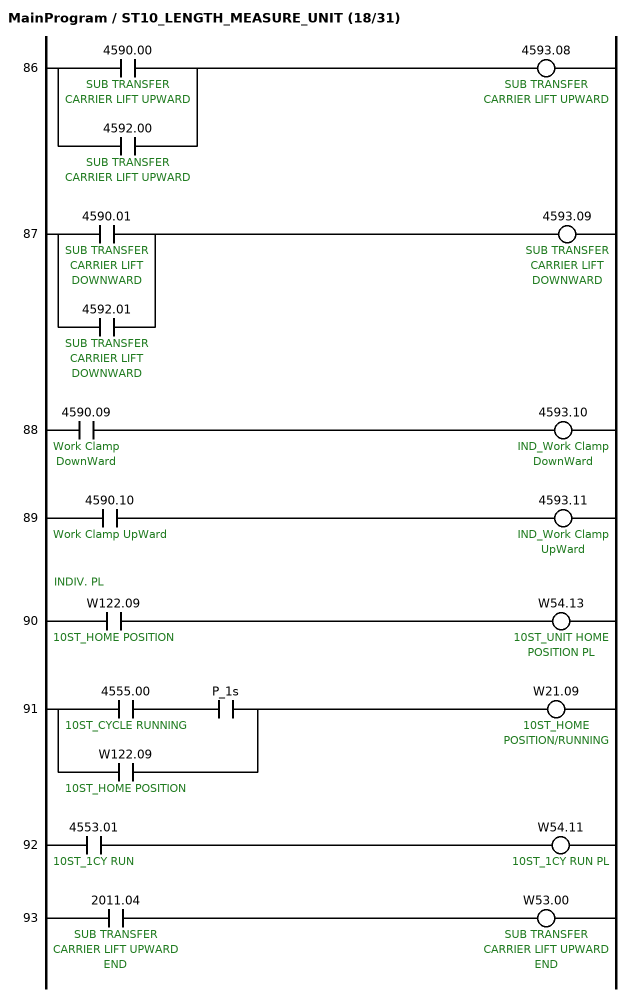
; [picture p504: MainProgram / ST10_LENGTH_MEASURE_UNIT, rungs 86-93]
; rung 86
LD 4590.00  ; SUB TRANSFER CARRIER LIFT UPWARD
OR 4592.00  ; SUB TRANSFER CARRIER LIFT UPWARD
OUT 4593.08  ; SUB TRANSFER CARRIER LIFT UPWARD
; rung 87
LD 4590.01  ; SUB TRANSFER CARRIER LIFT DOWNWARD
OR 4592.01  ; SUB TRANSFER CARRIER LIFT DOWNWARD
OUT 4593.09  ; SUB TRANSFER CARRIER LIFT DOWNWARD
; rung 88
LD 4590.09  ; Work Clamp DownWard
OUT 4593.10  ; IND_Work Clamp DownWard
; rung 89
LD 4590.10  ; Work Clamp UpWard
OUT 4593.11  ; IND_Work Clamp UpWard
; rung 90: INDIV. PL
LD W122.09  ; 10ST_HOME POSITION
OUT W54.13  ; 10ST_UNIT HOME POSITION PL
; rung 91
LD 4555.00  ; 10ST_CYCLE RUNNING
AND P_1s
OR W122.09  ; 10ST_HOME POSITION
OUT W21.09  ; 10ST_HOME POSITION/RUNNING
; rung 92
LD 4553.01  ; 10ST_1CY RUN
OUT W54.11  ; 10ST_1CY RUN PL
; rung 93
LD 2011.04  ; SUB TRANSFER CARRIER LIFT UPWARD END
OUT W53.00  ; SUB TRANSFER CARRIER LIFT UPWARD END

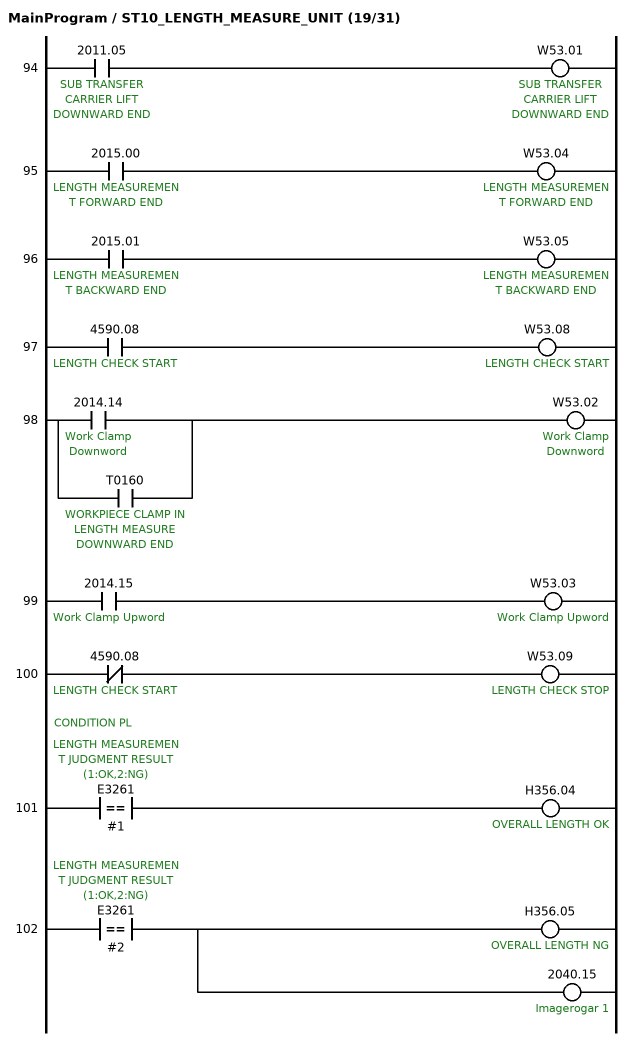
; rung 94
LD 2011.05  ; SUB TRANSFER CARRIER LIFT DOWNWARD END
OUT W53.01  ; SUB TRANSFER CARRIER LIFT DOWNWARD END
; rung 95
LD 2015.00  ; LENGTH MEASUREMENT FORWARD END
OUT W53.04  ; LENGTH MEASUREMENT FORWARD END
; rung 96
LD 2015.01  ; LENGTH MEASUREMENT BACKWARD END
OUT W53.05  ; LENGTH MEASUREMENT BACKWARD END
; rung 97
LD 4590.08  ; LENGTH CHECK START
OUT W53.08  ; LENGTH CHECK START
; rung 98
LD 2014.14  ; Work Clamp Downword
OR T0160  ; WORKPIECE CLAMP IN LENGTH MEASURE DOWNWARD END
OUT W53.02  ; Work Clamp Downword
; rung 99
LD 2014.15  ; Work Clamp Upword
OUT W53.03  ; Work Clamp Upword
; rung 100
LDNOT 4590.08  ; LENGTH CHECK START
OUT W53.09  ; LENGTH CHECK STOP
; rung 101: CONDITION PL
LD=(300) E3261 #1  ; LENGTH MEASUREMENT JUDGMENT RESULT (1:OK,2:NG)
OUT H356.04  ; OVERALL LENGTH OK
; rung 102
LD=(300) E3261 #2  ; LENGTH MEASUREMENT JUDGMENT RESULT (1:OK,2:NG)
OUT H356.05  ; OVERALL LENGTH NG
OUT 2040.15  ; Imagerogar 1

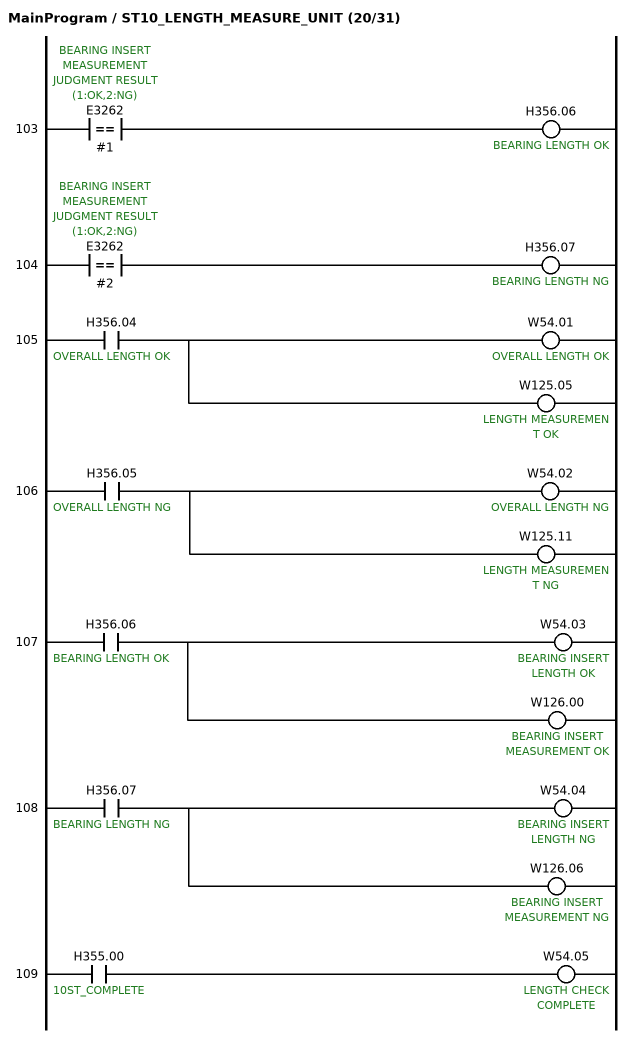
; rung 103
LD=(300) E3262 #1  ; BEARING INSERT MEASUREMENT  JUDGMENT RESULT (1:OK,2:NG)
OUT H356.06  ; BEARING LENGTH OK
; rung 104
LD=(300) E3262 #2  ; BEARING INSERT MEASUREMENT  JUDGMENT RESULT (1:OK,2:NG)
OUT H356.07  ; BEARING LENGTH NG
; rung 105
LD H356.04  ; OVERALL LENGTH OK
OUT W54.01  ; OVERALL LENGTH OK
OUT W125.05  ; LENGTH MEASUREMENT OK
; rung 106
LD H356.05  ; OVERALL LENGTH NG
OUT W54.02  ; OVERALL LENGTH NG
OUT W125.11  ; LENGTH MEASUREMENT NG
; rung 107
LD H356.06  ; BEARING LENGTH OK
OUT W54.03  ; BEARING INSERT LENGTH OK
OUT W126.00  ; BEARING INSERT MEASUREMENT OK
; rung 108
LD H356.07  ; BEARING LENGTH NG
OUT W54.04  ; BEARING INSERT LENGTH NG
OUT W126.06  ; BEARING INSERT MEASUREMENT NG
; rung 109
LD H355.00  ; 10ST_COMPLETE
OUT W54.05  ; LENGTH CHECK COMPLETE

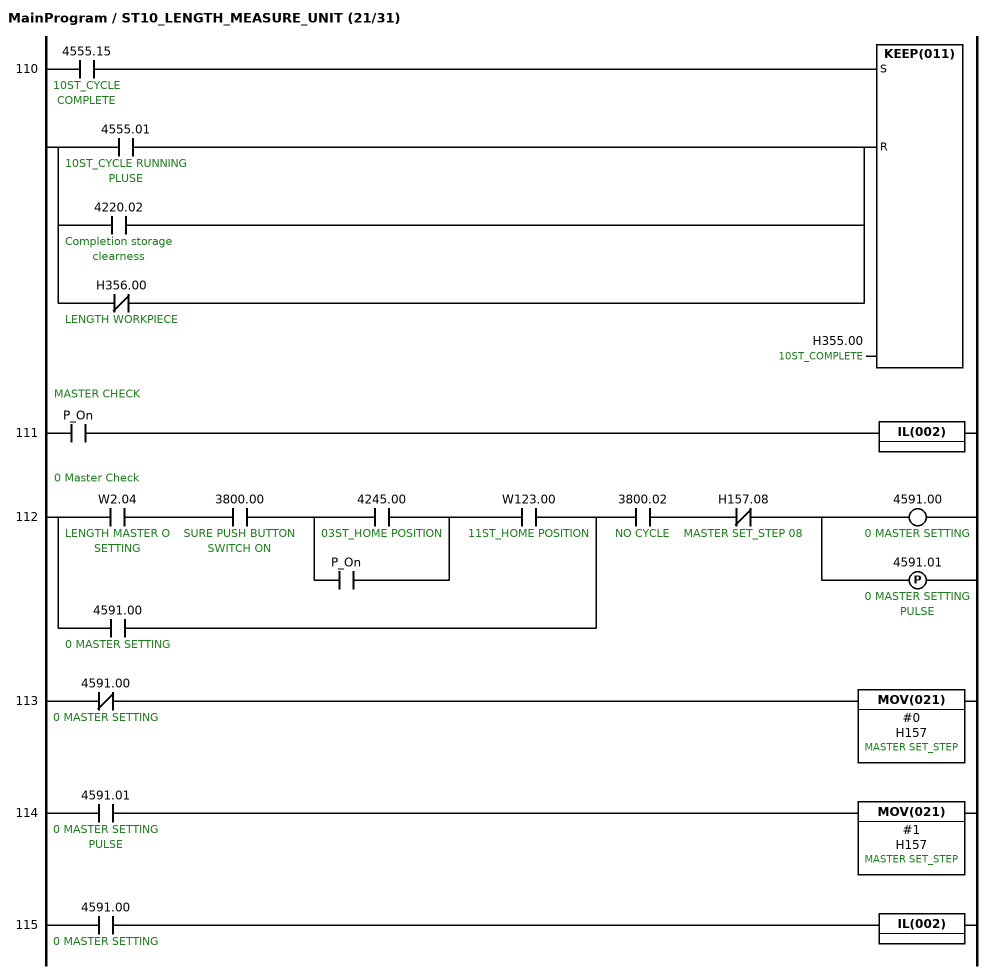
; rung 110
LD 4555.15  ; 10ST_CYCLE COMPLETE
LD 4555.01  ; 10ST_CYCLE RUNNING PLUSE
OR 4220.02  ; Completion storage clearness
ORNOT H356.00  ; LENGTH WORKPIECE
KEEP(011) H355.00  ; 10ST_COMPLETE
; rung 111: MASTER CHECK
LD P_On
IL(002)
; rung 112: 0 Master Check
LD W2.04  ; LENGTH MASTER O SETTING
AND 3800.00  ; SURE PUSH BUTTON SWITCH ON
LD 4245.00  ; 03ST_HOME POSITION
OR P_On
ANDLD
AND W123.00  ; 11ST_HOME POSITION
OR 4591.00  ; 0 MASTER SETTING
AND 3800.02  ; NO CYCLE
ANDNOT H157.08  ; MASTER SET_STEP 08
OUT 4591.00  ; 0 MASTER SETTING
DIFU(013) 4591.01  ; 0 MASTER SETTING PULSE
; rung 113
LDNOT 4591.00  ; 0 MASTER SETTING
MOV(021) #0 H157  ; MASTER SET_STEP
; rung 114
LD 4591.01  ; 0 MASTER SETTING PULSE
MOV(021) #1 H157  ; MASTER SET_STEP
; rung 115
LD 4591.00  ; 0 MASTER SETTING
IL(002)

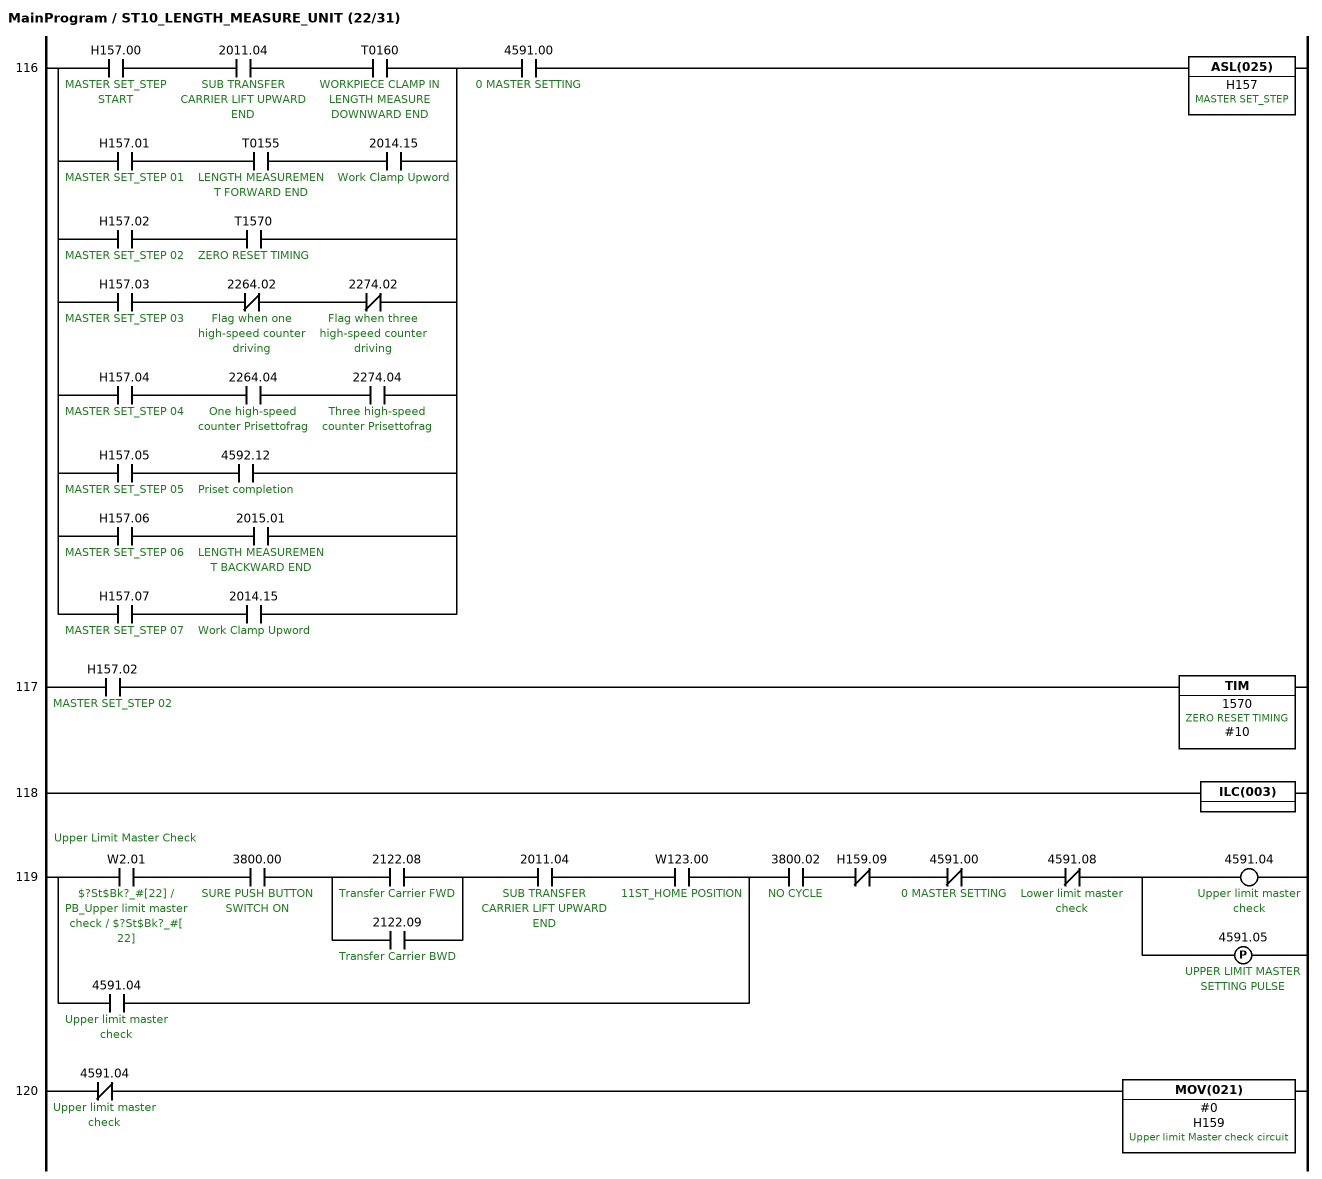
; rung 116
LD H157.00  ; MASTER SET_STEP START
AND 2011.04  ; SUB TRANSFER CARRIER LIFT UPWARD END
AND T0160  ; WORKPIECE CLAMP IN LENGTH MEASURE DOWNWARD END
LD H157.01  ; MASTER SET_STEP 01
AND T0155  ; LENGTH MEASUREMENT FORWARD END
AND 2014.15  ; Work Clamp Upword
ORLD
LD H157.02  ; MASTER SET_STEP 02
AND T1570  ; ZERO RESET TIMING
ORLD
LD H157.03  ; MASTER SET_STEP 03
ANDNOT 2264.02  ; Flag when one high-speed counter driving
ANDNOT 2274.02  ; Flag when three high-speed counter driving
ORLD
LD H157.04  ; MASTER SET_STEP 04
AND 2264.04  ; One high-speed counter Prisettofrag
AND 2274.04  ; Three high-speed counter Prisettofrag
ORLD
LD H157.05  ; MASTER SET_STEP 05
AND 4592.12  ; Priset completion
ORLD
LD H157.06  ; MASTER SET_STEP 06
AND 2015.01  ; LENGTH MEASUREMENT BACKWARD END
ORLD
LD H157.07  ; MASTER SET_STEP 07
AND 2014.15  ; Work Clamp Upword
ORLD
AND 4591.00  ; 0 MASTER SETTING
ASL(025) H157  ; MASTER SET_STEP
; rung 117
LD H157.02  ; MASTER SET_STEP 02
TIM 1570 #10  ; ZERO RESET TIMING
; rung 118
ILC(003)
; rung 119: Upper Limit Master Check
LD W2.01  ; $?St$Bk?_#[22] / PB_Upper limit master check / $?St$Bk?_#[22]
AND 3800.00  ; SURE PUSH BUTTON SWITCH ON
LD 2122.08  ; Transfer Carrier FWD
OR 2122.09  ; Transfer Carrier BWD
ANDLD
AND 2011.04  ; SUB TRANSFER CARRIER LIFT UPWARD END
AND W123.00  ; 11ST_HOME POSITION
OR 4591.04  ; Upper limit master check
AND 3800.02  ; NO CYCLE
ANDNOT H159.09
ANDNOT 4591.00  ; 0 MASTER SETTING
ANDNOT 4591.08  ; Lower limit master check
OUT 4591.04  ; Upper limit master check
DIFU(013) 4591.05  ; UPPER LIMIT MASTER SETTING PULSE
; rung 120
LDNOT 4591.04  ; Upper limit master check
MOV(021) #0 H159  ; Upper limit Master check circuit

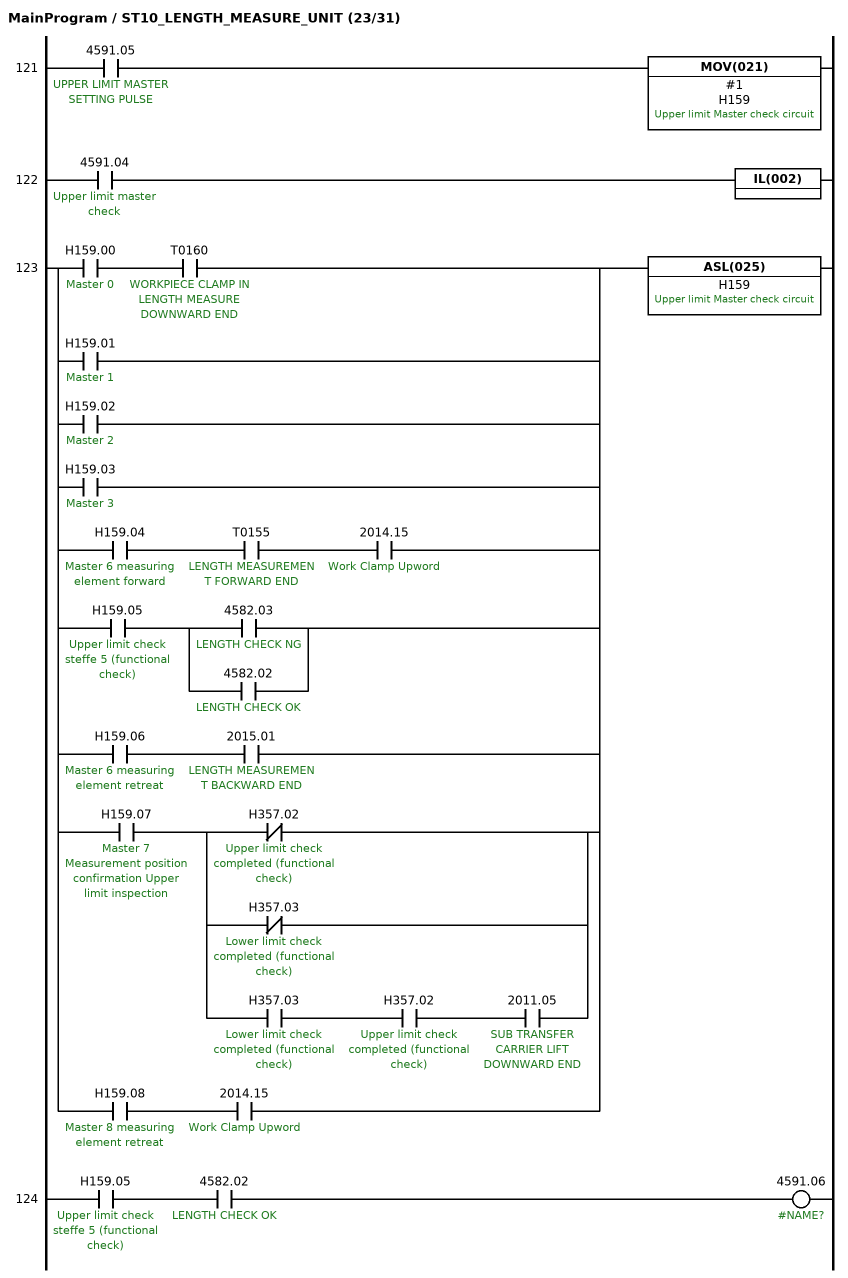
; rung 121
LD 4591.05  ; UPPER LIMIT MASTER SETTING PULSE
MOV(021) #1 H159  ; Upper limit Master check circuit
; rung 122
LD 4591.04  ; Upper limit master check
IL(002)
; rung 123
LD H159.00  ; Master 0
AND T0160  ; WORKPIECE CLAMP IN LENGTH MEASURE DOWNWARD END
OR H159.01  ; Master 1
OR H159.02  ; Master 2
OR H159.03  ; Master 3
LD H159.04  ; Master 6 measuring element forward
AND T0155  ; LENGTH MEASUREMENT FORWARD END
AND 2014.15  ; Work Clamp Upword
ORLD
LD H159.05  ; Upper limit check steffe 5 (functional check)
LD 4582.03  ; LENGTH CHECK NG
OR 4582.02  ; LENGTH CHECK OK
ANDLD
ORLD
LD H159.06  ; Master 6 measuring element retreat
AND 2015.01  ; LENGTH MEASUREMENT BACKWARD END
ORLD
LD H159.07  ; Master 7 Measurement position confirmation Upper limit inspection
LDNOT H357.02  ; Upper limit check completed (functional check)
ORNOT H357.03  ; Lower limit check completed (functional check)
LD H357.03  ; Lower limit check completed (functional check)
AND H357.02  ; Upper limit check completed (functional check)
AND 2011.05  ; SUB TRANSFER CARRIER LIFT DOWNWARD END
ORLD
ANDLD
ORLD
LD H159.08  ; Master 8 measuring element retreat
AND 2014.15  ; Work Clamp Upword
ORLD
ASL(025) H159  ; Upper limit Master check circuit
; rung 124
LD H159.05  ; Upper limit check steffe 5 (functional check)
AND 4582.02  ; LENGTH CHECK OK
OUT 4591.06  ; #NAME?

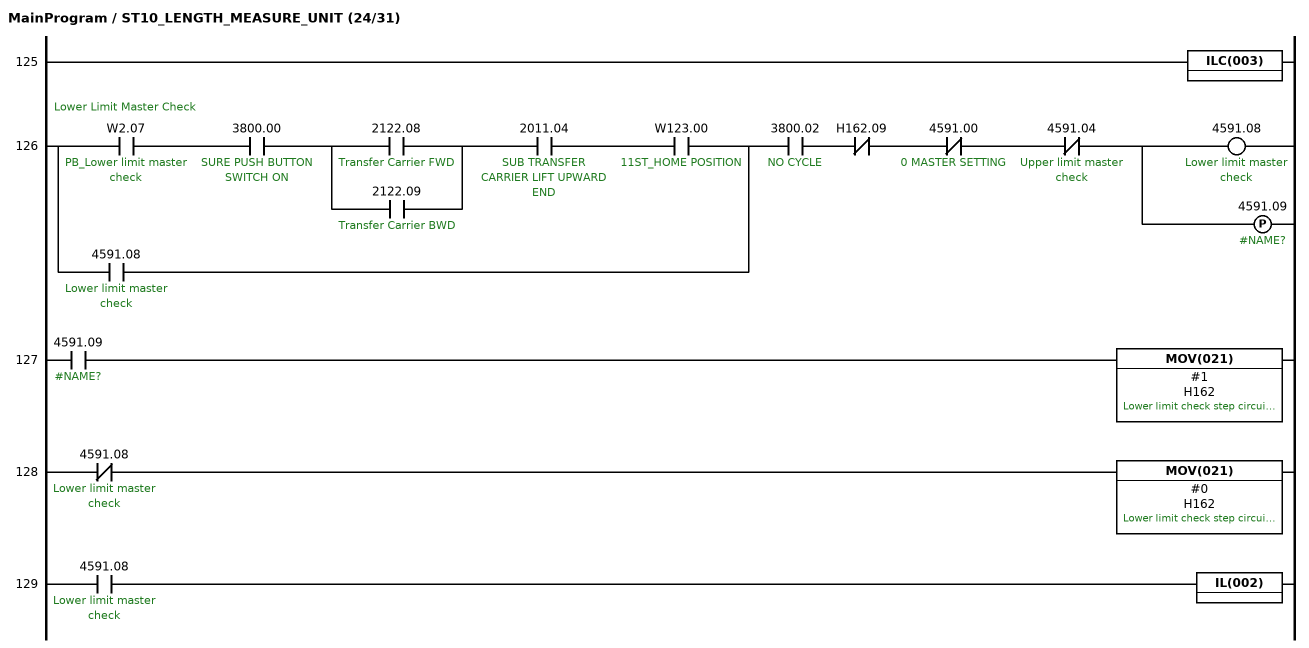
; rung 125
ILC(003)
; rung 126: Lower Limit Master Check
LD W2.07  ; PB_Lower limit master check
AND 3800.00  ; SURE PUSH BUTTON SWITCH ON
LD 2122.08  ; Transfer Carrier FWD
OR 2122.09  ; Transfer Carrier BWD
ANDLD
AND 2011.04  ; SUB TRANSFER CARRIER LIFT UPWARD END
AND W123.00  ; 11ST_HOME POSITION
OR 4591.08  ; Lower limit master check
AND 3800.02  ; NO CYCLE
ANDNOT H162.09
ANDNOT 4591.00  ; 0 MASTER SETTING
ANDNOT 4591.04  ; Upper limit master check
OUT 4591.08  ; Lower limit master check
DIFU(013) 4591.09  ; #NAME?
; rung 127
LD 4591.09  ; #NAME?
MOV(021) #1 H162  ; Lower limit check step circuit (functional check)
; rung 128
LDNOT 4591.08  ; Lower limit master check
MOV(021) #0 H162  ; Lower limit check step circuit (functional check)
; rung 129
LD 4591.08  ; Lower limit master check
IL(002)

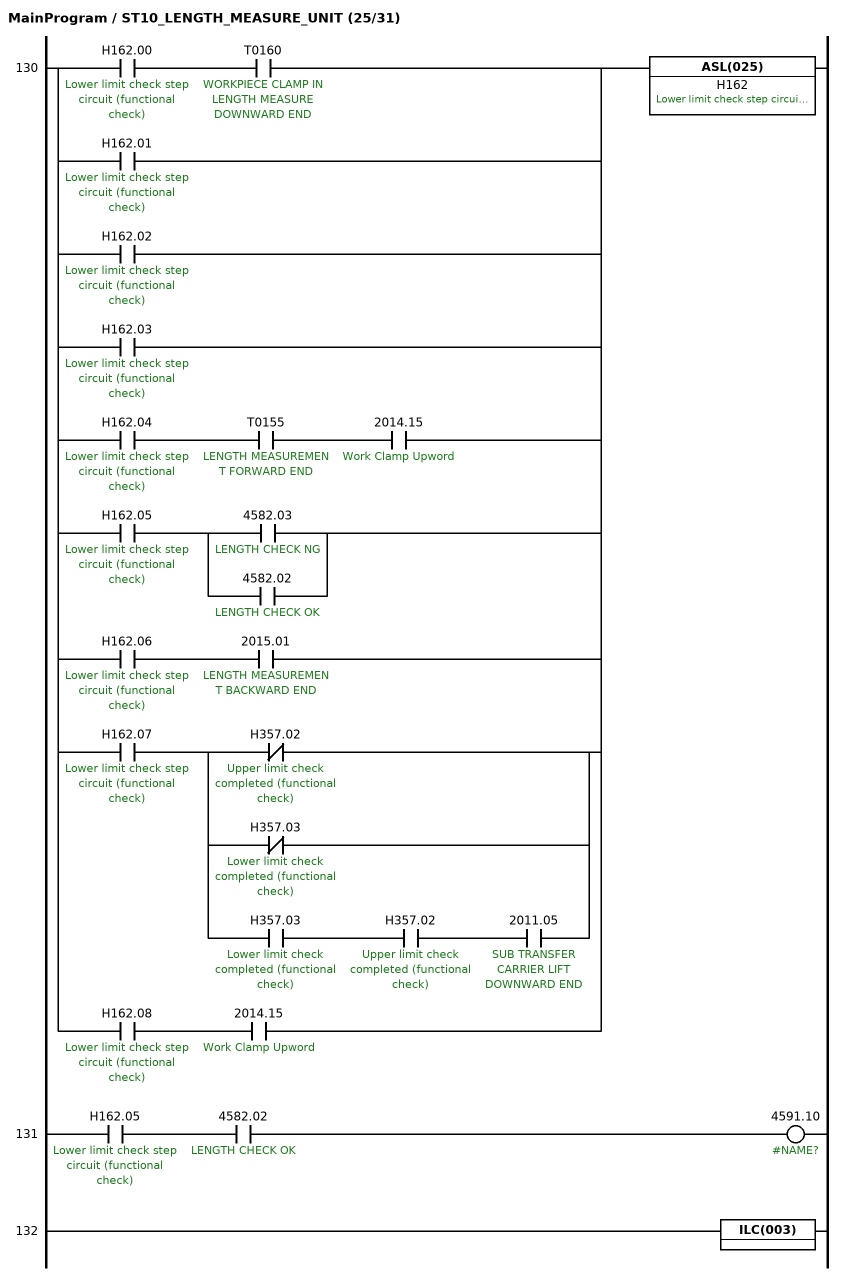
; rung 130
LD H162.00  ; Lower limit check step circuit (functional check)
AND T0160  ; WORKPIECE CLAMP IN LENGTH MEASURE DOWNWARD END
OR H162.01  ; Lower limit check step circuit (functional check)
OR H162.02  ; Lower limit check step circuit (functional check)
OR H162.03  ; Lower limit check step circuit (functional check)
LD H162.04  ; Lower limit check step circuit (functional check)
AND T0155  ; LENGTH MEASUREMENT FORWARD END
AND 2014.15  ; Work Clamp Upword
ORLD
LD H162.05  ; Lower limit check step circuit (functional check)
LD 4582.03  ; LENGTH CHECK NG
OR 4582.02  ; LENGTH CHECK OK
ANDLD
ORLD
LD H162.06  ; Lower limit check step circuit (functional check)
AND 2015.01  ; LENGTH MEASUREMENT BACKWARD END
ORLD
LD H162.07  ; Lower limit check step circuit (functional check)
LDNOT H357.02  ; Upper limit check completed (functional check)
ORNOT H357.03  ; Lower limit check completed (functional check)
LD H357.03  ; Lower limit check completed (functional check)
AND H357.02  ; Upper limit check completed (functional check)
AND 2011.05  ; SUB TRANSFER CARRIER LIFT DOWNWARD END
ORLD
ANDLD
ORLD
LD H162.08  ; Lower limit check step circuit (functional check)
AND 2014.15  ; Work Clamp Upword
ORLD
ASL(025) H162  ; Lower limit check step circuit (functional check)
; rung 131
LD H162.05  ; Lower limit check step circuit (functional check)
AND 4582.02  ; LENGTH CHECK OK
OUT 4591.10  ; #NAME?
; rung 132
ILC(003)

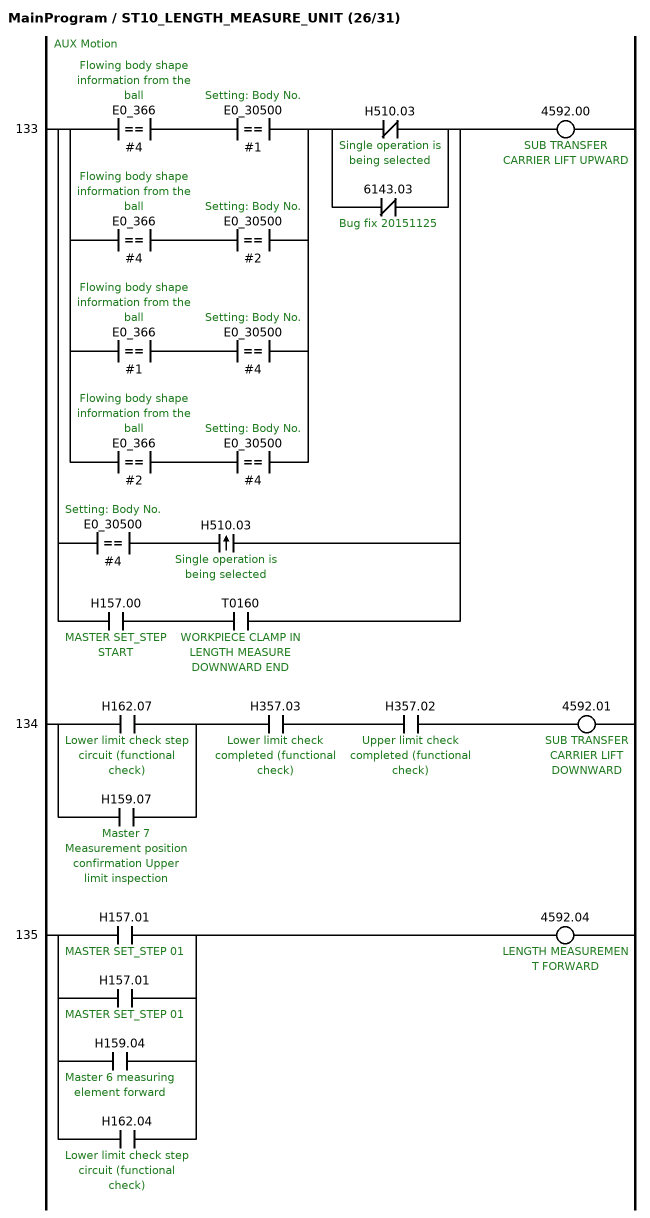
; rung 133: AUX Motion
LD=(300) E0_366 #4  ; Flowing body shape information from the ball
AND=(300) E0_30500 #1  ; Setting: Body No.
LD=(300) E0_366 #4  ; Flowing body shape information from the ball
AND=(300) E0_30500 #2  ; Setting: Body No.
ORLD
LD=(300) E0_366 #1  ; Flowing body shape information from the ball
AND=(300) E0_30500 #4  ; Setting: Body No.
ORLD
LD=(300) E0_366 #2  ; Flowing body shape information from the ball
AND=(300) E0_30500 #4  ; Setting: Body No.
ORLD
LDNOT H510.03  ; Single operation is being selected
ORNOT 6143.03  ; Bug fix 20151125
ANDLD
LD=(300) E0_30500 #4  ; Setting: Body No.
@AND H510.03  ; Single operation is being selected
ORLD
LD H157.00  ; MASTER SET_STEP START
AND T0160  ; WORKPIECE CLAMP IN LENGTH MEASURE DOWNWARD END
ORLD
OUT 4592.00  ; SUB TRANSFER CARRIER LIFT UPWARD
; rung 134
LD H162.07  ; Lower limit check step circuit (functional check)
OR H159.07  ; Master 7 Measurement position confirmation Upper limit inspection
AND H357.03  ; Lower limit check completed (functional check)
AND H357.02  ; Upper limit check completed (functional check)
OUT 4592.01  ; SUB TRANSFER CARRIER LIFT DOWNWARD
; rung 135
LD H157.01  ; MASTER SET_STEP 01
OR H157.01  ; MASTER SET_STEP 01
OR H159.04  ; Master 6 measuring element forward
OR H162.04  ; Lower limit check step circuit (functional check)
OUT 4592.04  ; LENGTH MEASUREMENT FORWARD

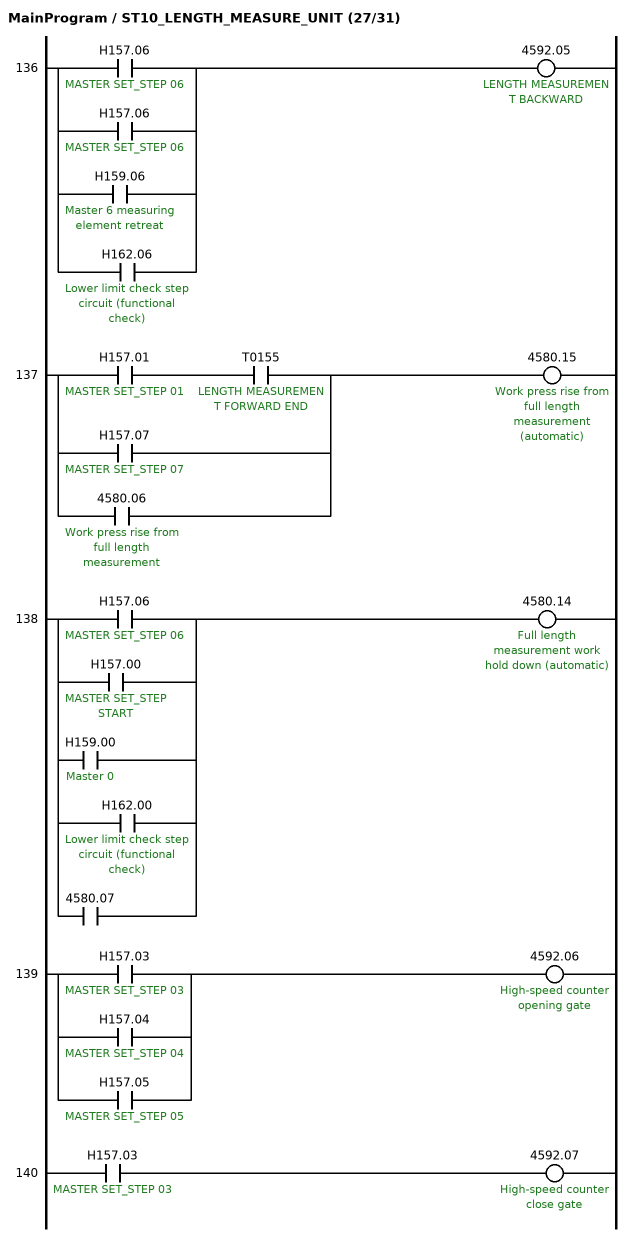
; rung 136
LD H157.06  ; MASTER SET_STEP 06
OR H157.06  ; MASTER SET_STEP 06
OR H159.06  ; Master 6 measuring element retreat
OR H162.06  ; Lower limit check step circuit (functional check)
OUT 4592.05  ; LENGTH MEASUREMENT BACKWARD
; rung 137
LD H157.01  ; MASTER SET_STEP 01
AND T0155  ; LENGTH MEASUREMENT FORWARD END
OR H157.07  ; MASTER SET_STEP 07
OR 4580.06  ; Work press rise from full length measurement
OUT 4580.15  ; Work press rise from full length measurement (automatic)
; rung 138
LD H157.06  ; MASTER SET_STEP 06
OR H157.00  ; MASTER SET_STEP START
OR H159.00  ; Master 0
OR H162.00  ; Lower limit check step circuit (functional check)
OR 4580.07
OUT 4580.14  ; Full length measurement work hold down (automatic)
; rung 139
LD H157.03  ; MASTER SET_STEP 03
OR H157.04  ; MASTER SET_STEP 04
OR H157.05  ; MASTER SET_STEP 05
OUT 4592.06  ; High-speed counter opening gate
; rung 140
LD H157.03  ; MASTER SET_STEP 03
OUT 4592.07  ; High-speed counter close gate

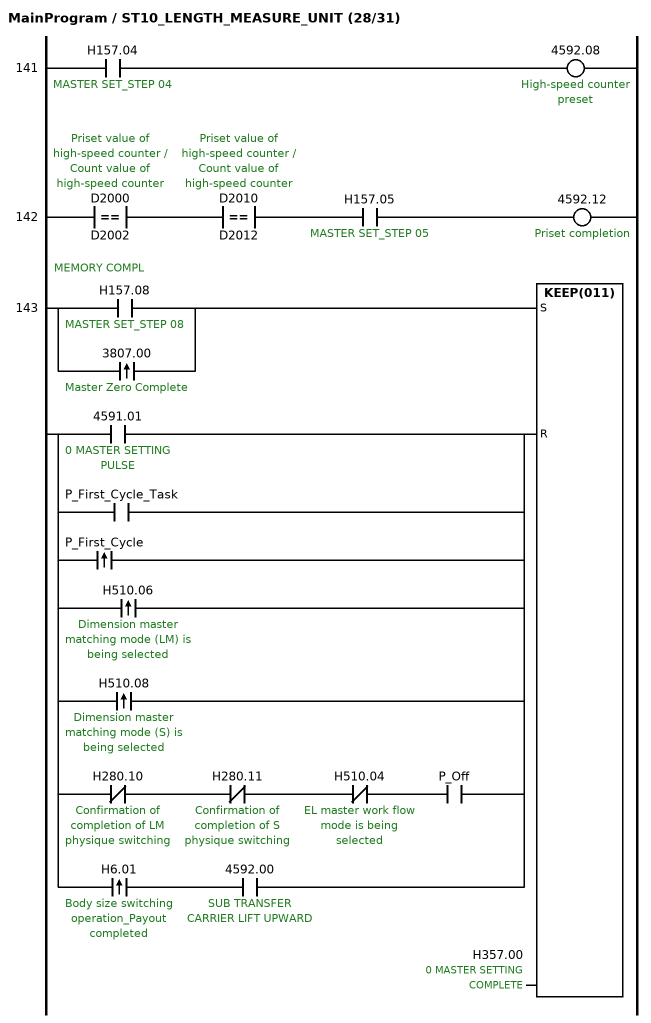
; rung 141
LD H157.04  ; MASTER SET_STEP 04
OUT 4592.08  ; High-speed counter preset
; rung 142
LD=SL(303) D2000 D2002  ; Priset value of high-speed counter, Count value of high-speed counter
AND=SL(303) D2010 D2012  ; Priset value of high-speed counter, Count value of high-speed counter
AND H157.05  ; MASTER SET_STEP 05
OUT 4592.12  ; Priset completion
; rung 143: MEMORY COMPL
LD H157.08  ; MASTER SET_STEP 08
@OR 3807.00  ; Master Zero Complete
LD 4591.01  ; 0 MASTER SETTING PULSE
OR P_First_Cycle_Task
@OR P_First_Cycle
@OR H510.06  ; Dimension master matching mode (LM) is being selected
@OR H510.08  ; Dimension master matching mode (S) is being selected
LDNOT H280.10  ; Confirmation of completion of LM physique switching
ANDNOT H280.11  ; Confirmation of completion of S physique switching
ANDNOT H510.04  ; EL master work flow mode is being selected
AND P_Off
ORLD
@LD H6.01  ; Body size switching operation_Payout completed
AND 4592.00  ; SUB TRANSFER CARRIER LIFT UPWARD
ORLD
KEEP(011) H357.00  ; 0 MASTER SETTING COMPLETE

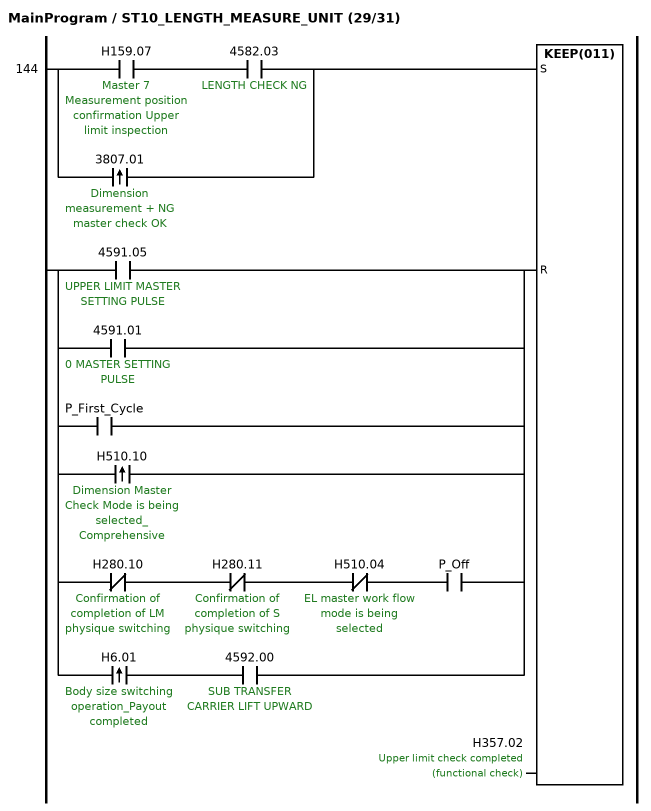
; rung 144
LD H159.07  ; Master 7 Measurement position confirmation Upper limit inspection
AND 4582.03  ; LENGTH CHECK NG
@OR 3807.01  ; Dimension measurement + NG master check OK
LD 4591.05  ; UPPER LIMIT MASTER SETTING PULSE
OR 4591.01  ; 0 MASTER SETTING PULSE
OR P_First_Cycle
@OR H510.10  ; Dimension Master Check Mode is being selected_Comprehensive
LDNOT H280.10  ; Confirmation of completion of LM physique switching
ANDNOT H280.11  ; Confirmation of completion of S physique switching
ANDNOT H510.04  ; EL master work flow mode is being selected
AND P_Off
ORLD
@LD H6.01  ; Body size switching operation_Payout completed
AND 4592.00  ; SUB TRANSFER CARRIER LIFT UPWARD
ORLD
KEEP(011) H357.02  ; Upper limit check completed (functional check)

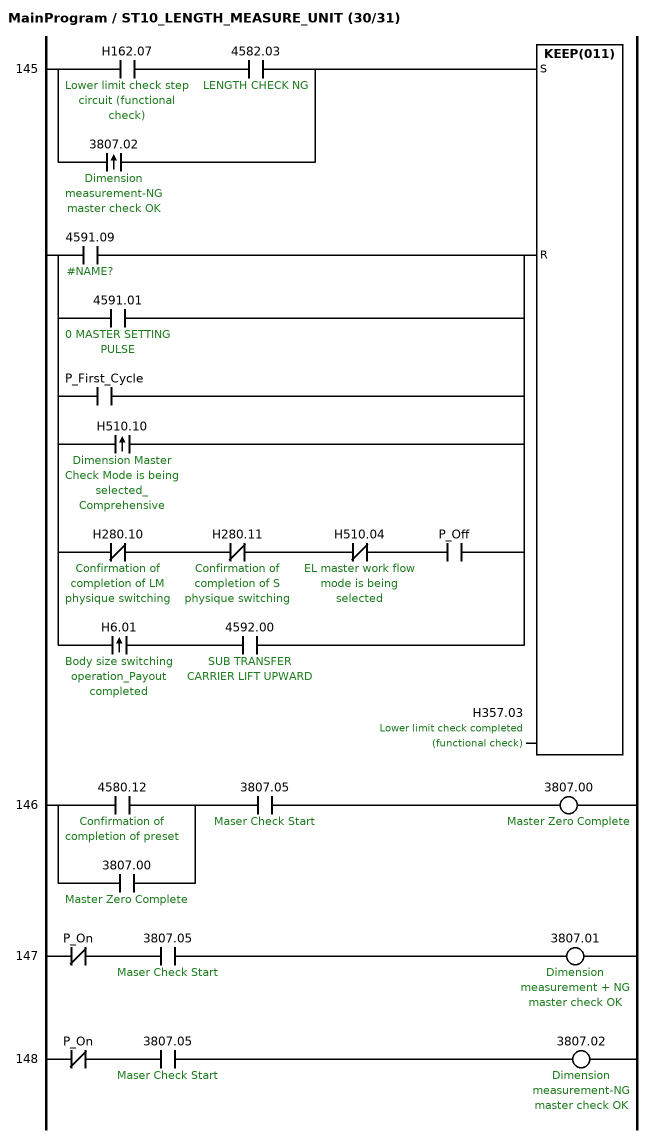
; rung 145
LD H162.07  ; Lower limit check step circuit (functional check)
AND 4582.03  ; LENGTH CHECK NG
@OR 3807.02  ; Dimension measurement-NG master check OK
LD 4591.09  ; #NAME?
OR 4591.01  ; 0 MASTER SETTING PULSE
OR P_First_Cycle
@OR H510.10  ; Dimension Master Check Mode is being selected_Comprehensive
LDNOT H280.10  ; Confirmation of completion of LM physique switching
ANDNOT H280.11  ; Confirmation of completion of S physique switching
ANDNOT H510.04  ; EL master work flow mode is being selected
AND P_Off
ORLD
@LD H6.01  ; Body size switching operation_Payout completed
AND 4592.00  ; SUB TRANSFER CARRIER LIFT UPWARD
ORLD
KEEP(011) H357.03  ; Lower limit check completed (functional check)
; rung 146
LD 4580.12  ; Confirmation of completion of preset
OR 3807.00  ; Master Zero Complete
AND 3807.05  ; Maser Check Start
OUT 3807.00  ; Master Zero Complete
; rung 147
LDNOT P_On
AND 3807.05  ; Maser Check Start
OUT 3807.01  ; Dimension measurement + NG master check OK
; rung 148
LDNOT P_On
AND 3807.05  ; Maser Check Start
OUT 3807.02  ; Dimension measurement-NG master check OK

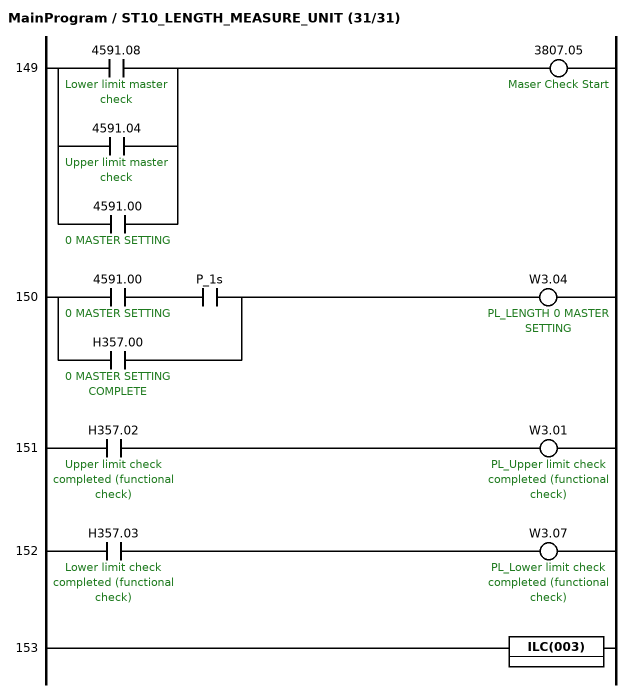
; rung 149
LD 4591.08  ; Lower limit master check
OR 4591.04  ; Upper limit master check
OR 4591.00  ; 0 MASTER SETTING
OUT 3807.05  ; Maser Check Start
; rung 150
LD 4591.00  ; 0 MASTER SETTING
AND P_1s
OR H357.00  ; 0 MASTER SETTING COMPLETE
OUT W3.04  ; PL_LENGTH 0 MASTER SETTING
; rung 151
LD H357.02  ; Upper limit check completed (functional check)
OUT W3.01  ; PL_Upper limit check completed (functional check)
; rung 152
LD H357.03  ; Lower limit check completed (functional check)
OUT W3.07  ; PL_Lower limit check completed (functional check)
; rung 153
ILC(003)

### Section ST11_UNLOADING_UNIT

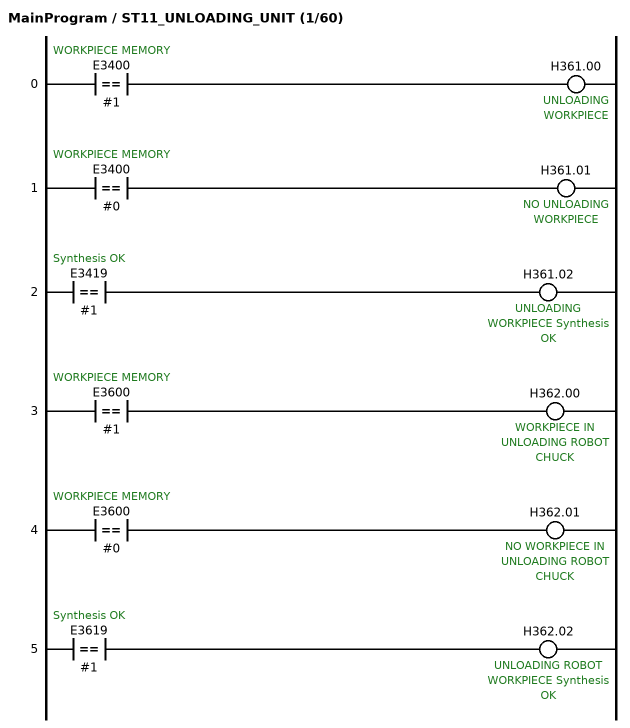
; rung 0
LD=(300) E3400 #1  ; WORKPIECE MEMORY
OUT H361.00  ; UNLOADING WORKPIECE
; rung 1
LD=(300) E3400 #0  ; WORKPIECE MEMORY
OUT H361.01  ; NO UNLOADING WORKPIECE
; rung 2
LD=(300) E3419 #1  ; Synthesis OK
OUT H361.02  ; UNLOADING WORKPIECE Synthesis OK
; rung 3
LD=(300) E3600 #1  ; WORKPIECE MEMORY
OUT H362.00  ; WORKPIECE IN UNLOADING ROBOT CHUCK
; rung 4
LD=(300) E3600 #0  ; WORKPIECE MEMORY
OUT H362.01  ; NO WORKPIECE IN UNLOADING ROBOT CHUCK
; rung 5
LD=(300) E3619 #1  ; Synthesis OK
OUT H362.02  ; UNLOADING ROBOT WORKPIECE Synthesis OK

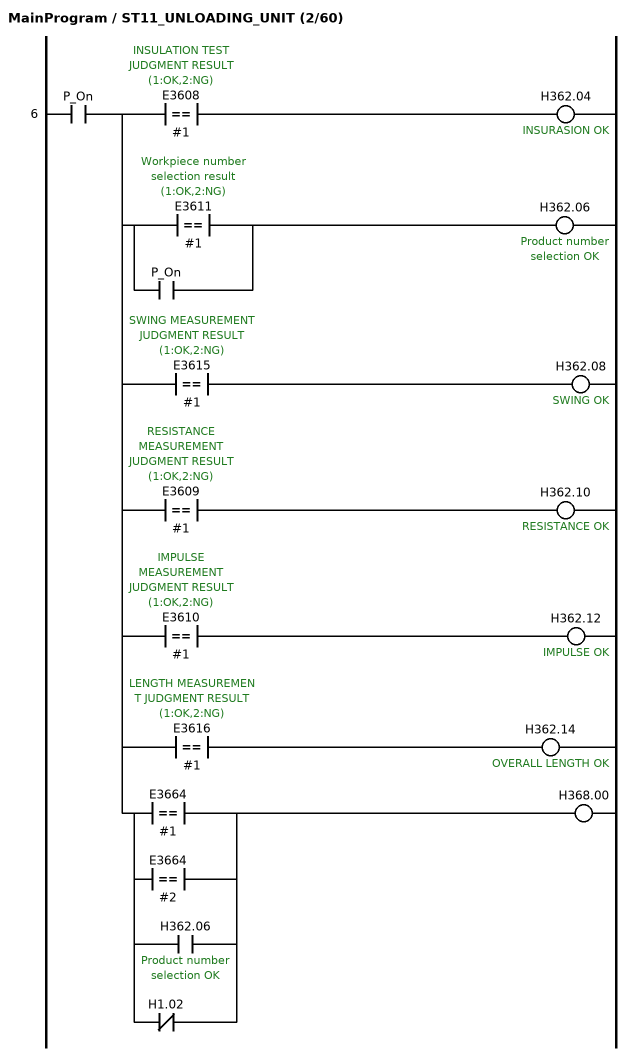
; rung 6
LD P_On
OUT TR0
AND=(300) E3608 #1  ; INSULATION TEST JUDGMENT RESULT (1:OK,2:NG)
OUT H362.04  ; INSURASION OK
LD TR0
LD=(300) E3611 #1  ; Workpiece number selection result (1:OK,2:NG)
OR P_On
ANDLD
OUT H362.06  ; Product number selection OK
LD TR0
AND=(300) E3615 #1  ; SWING MEASUREMENT JUDGMENT RESULT (1:OK,2:NG)
OUT H362.08  ; SWING OK
LD TR0
AND=(300) E3609 #1  ; RESISTANCE MEASUREMENT JUDGMENT RESULT (1:OK,2:NG)
OUT H362.10  ; RESISTANCE OK
LD TR0
AND=(300) E3610 #1  ; IMPULSE MEASUREMENT JUDGMENT RESULT (1:OK,2:NG)
OUT H362.12  ; IMPULSE OK
LD TR0
AND=(300) E3616 #1  ; LENGTH MEASUREMENT JUDGMENT RESULT (1:OK,2:NG)
OUT H362.14  ; OVERALL LENGTH OK
LD TR0
LD=(300) E3664 #1
OR=(300) E3664 #2
OR H362.06  ; Product number selection OK
ORNOT H1.02
ANDLD
OUT H368.00

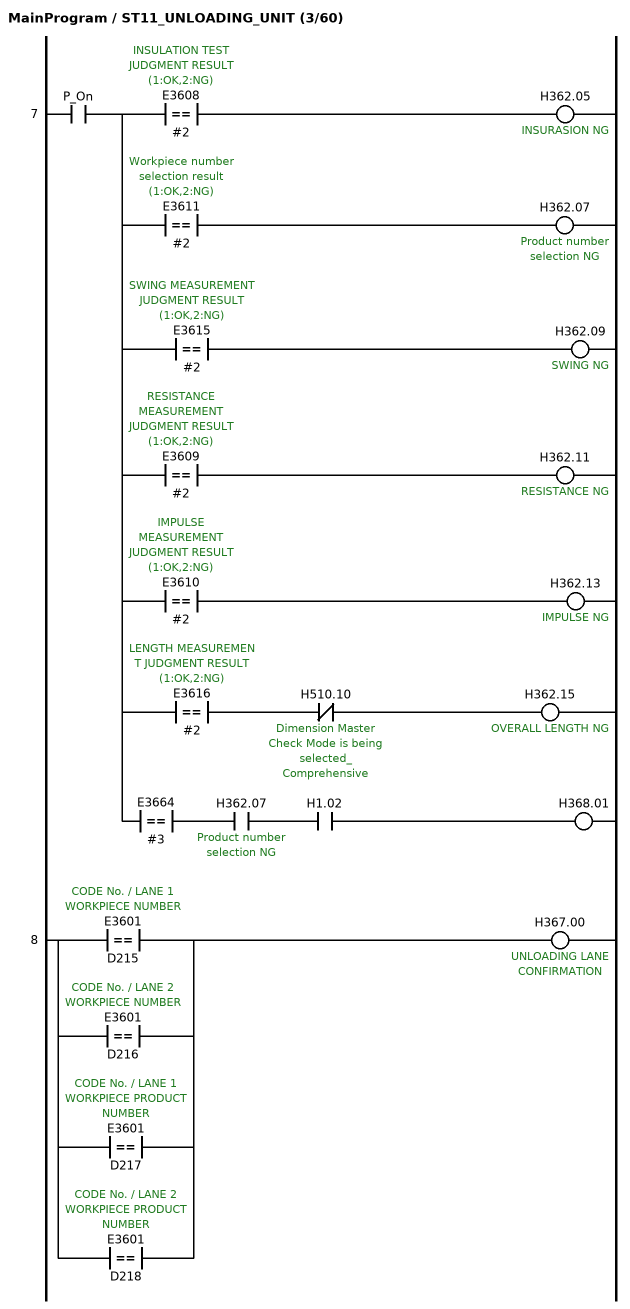
; rung 7
LD P_On
OUT TR0
AND=(300) E3608 #2  ; INSULATION TEST JUDGMENT RESULT (1:OK,2:NG)
OUT H362.05  ; INSURASION NG
LD TR0
AND=(300) E3611 #2  ; Workpiece number selection result (1:OK,2:NG)
OUT H362.07  ; Product number selection NG
LD TR0
AND=(300) E3615 #2  ; SWING MEASUREMENT JUDGMENT RESULT (1:OK,2:NG)
OUT H362.09  ; SWING NG
LD TR0
AND=(300) E3609 #2  ; RESISTANCE MEASUREMENT JUDGMENT RESULT (1:OK,2:NG)
OUT H362.11  ; RESISTANCE NG
LD TR0
AND=(300) E3610 #2  ; IMPULSE MEASUREMENT JUDGMENT RESULT (1:OK,2:NG)
OUT H362.13  ; IMPULSE NG
LD TR0
AND=(300) E3616 #2  ; LENGTH MEASUREMENT JUDGMENT RESULT (1:OK,2:NG)
ANDNOT H510.10  ; Dimension Master Check Mode is being selected_Comprehensive
OUT H362.15  ; OVERALL LENGTH NG
LD TR0
AND=(300) E3664 #3
AND H362.07  ; Product number selection NG
AND H1.02
OUT H368.01
; rung 8
LD=(300) E3601 D215  ; CODE No., LANE 1 WORKPIECE NUMBER
OR=(300) E3601 D216  ; CODE No., LANE 2 WORKPIECE NUMBER
OR=(300) E3601 D217  ; CODE No., LANE 1 WORKPIECE PRODUCT NUMBER
OR=(300) E3601 D218  ; CODE No., LANE 2 WORKPIECE PRODUCT NUMBER
OUT H367.00  ; UNLOADING LANE CONFIRMATION

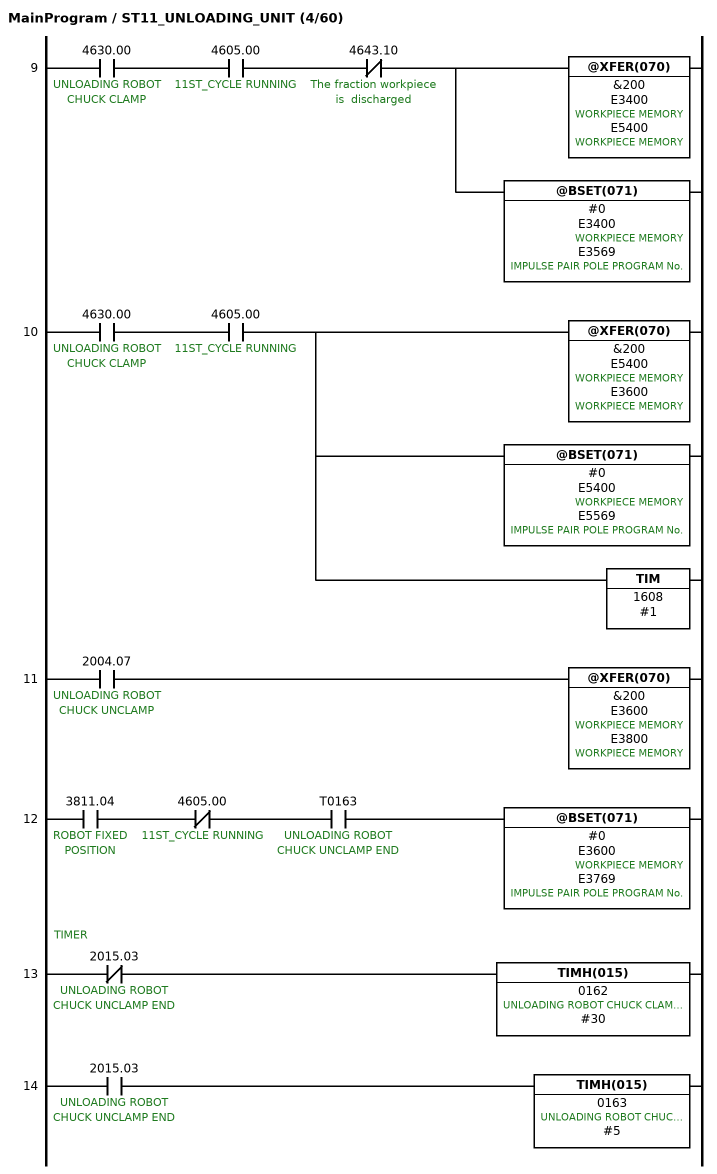
; rung 9
LD 4630.00  ; UNLOADING ROBOT CHUCK CLAMP
AND 4605.00  ; 11ST_CYCLE RUNNING
ANDNOT 4643.10  ; The fraction workpiece is  discharged
@XFER(070) &200 E3400 E5400  ; WORKPIECE MEMORY
@BSET(071) #0 E3400 E3569  ; WORKPIECE MEMORY, IMPULSE PAIR POLE PROGRAM No.
; rung 10
LD 4630.00  ; UNLOADING ROBOT CHUCK CLAMP
AND 4605.00  ; 11ST_CYCLE RUNNING
@XFER(070) &200 E5400 E3600  ; WORKPIECE MEMORY
@BSET(071) #0 E5400 E5569  ; WORKPIECE MEMORY, IMPULSE PAIR POLE PROGRAM No.
TIM 1608 #1
; rung 11
LD 2004.07  ; UNLOADING ROBOT CHUCK UNCLAMP
@XFER(070) &200 E3600 E3800  ; WORKPIECE MEMORY
; rung 12
LD 3811.04  ; ROBOT FIXED POSITION
ANDNOT 4605.00  ; 11ST_CYCLE RUNNING
AND T0163  ; UNLOADING ROBOT CHUCK UNCLAMP END
@BSET(071) #0 E3600 E3769  ; WORKPIECE MEMORY, IMPULSE PAIR POLE PROGRAM No.
; rung 13: TIMER
LDNOT 2015.03  ; UNLOADING ROBOT CHUCK UNCLAMP END
TIMH(015) 0162 #30  ; UNLOADING ROBOT CHUCK CLAMP END
; rung 14
LD 2015.03  ; UNLOADING ROBOT CHUCK UNCLAMP END
TIMH(015) 0163 #5  ; UNLOADING ROBOT CHUCK UNCLAMP END

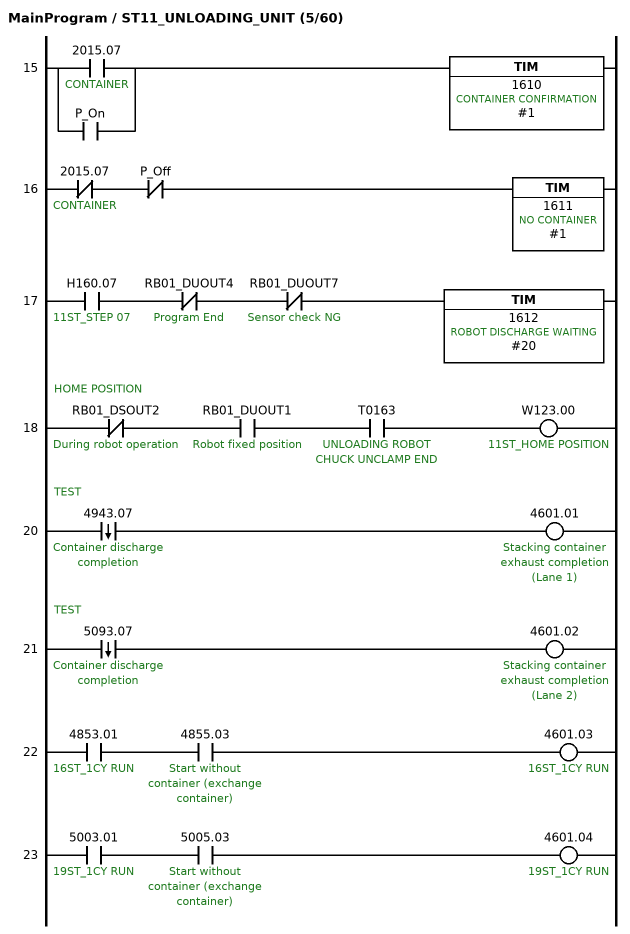
; rung 15
LD 2015.07  ; CONTAINER
OR P_On
TIM 1610 #1  ; CONTAINER CONFIRMATION
; rung 16
LDNOT 2015.07  ; CONTAINER
ANDNOT P_Off
TIM 1611 #1  ; NO CONTAINER
; rung 17
LD H160.07  ; 11ST_STEP 07
ANDNOT RB01_DUOUT4  ; Program End
ANDNOT RB01_DUOUT7  ; Sensor check NG
TIM 1612 #20  ; ROBOT DISCHARGE WAITING
; rung 18: HOME POSITION
LDNOT RB01_DSOUT2  ; During robot operation
AND RB01_DUOUT1  ; Robot fixed position
AND T0163  ; UNLOADING ROBOT CHUCK UNCLAMP END
OUT W123.00  ; 11ST_HOME POSITION
; rung 19: INTERFERENCE
; rung 20: TEST
%LD 4943.07  ; Container discharge completion
OUT 4601.01  ; Stacking container exhaust completion (Lane 1)
; rung 21: TEST
%LD 5093.07  ; Container discharge completion
OUT 4601.02  ; Stacking container exhaust completion (Lane 2)
; rung 22
LD 4853.01  ; 16ST_1CY RUN
AND 4855.03  ; Start without container (exchange container)
OUT 4601.03  ; 16ST_1CY RUN
; rung 23
LD 5003.01  ; 19ST_1CY RUN
AND 5005.03  ; Start without container (exchange container)
OUT 4601.04  ; 19ST_1CY RUN

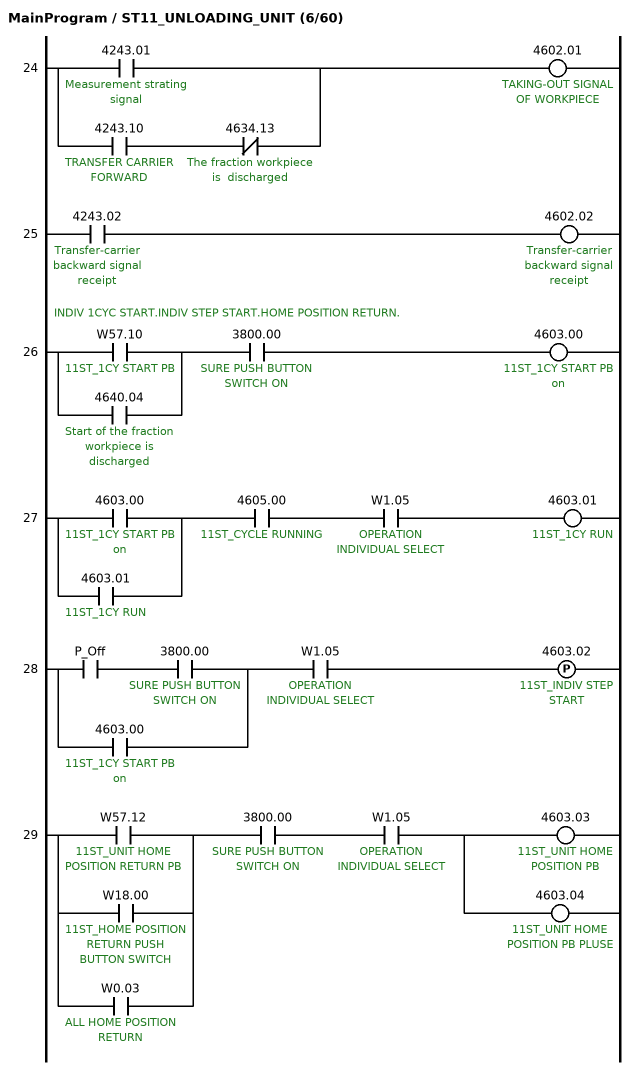
; rung 24
LD 4243.01  ; Measurement strating signal
LD 4243.10  ; TRANSFER CARRIER FORWARD
ANDNOT 4634.13  ; The fraction workpiece is  discharged
ORLD
OUT 4602.01  ; TAKING-OUT SIGNAL OF WORKPIECE
; rung 25
LD 4243.02  ; Transfer-carrier backward signal receipt
OUT 4602.02  ; Transfer-carrier backward signal receipt
; rung 26: INDIV 1CYC START.INDIV STEP START.HOME POSITION RETURN.
LD W57.10  ; 11ST_1CY START PB
OR 4640.04  ; Start of the fraction workpiece is discharged
AND 3800.00  ; SURE PUSH BUTTON SWITCH ON
OUT 4603.00  ; 11ST_1CY START PB on
; rung 27
LD 4603.00  ; 11ST_1CY START PB on
OR 4603.01  ; 11ST_1CY RUN
AND 4605.00  ; 11ST_CYCLE RUNNING
AND W1.05  ; OPERATION INDIVIDUAL SELECT
OUT 4603.01  ; 11ST_1CY RUN
; rung 28
LD P_Off
AND 3800.00  ; SURE PUSH BUTTON SWITCH ON
OR 4603.00  ; 11ST_1CY START PB on
AND W1.05  ; OPERATION INDIVIDUAL SELECT
DIFU(013) 4603.02  ; 11ST_INDIV STEP START
; rung 29
LD W57.12  ; 11ST_UNIT HOME POSITION RETURN PB
OR W18.00  ; 11ST_HOME POSITION RETURN PUSH BUTTON SWITCH
OR W0.03  ; ALL HOME POSITION RETURN
AND 3800.00  ; SURE PUSH BUTTON SWITCH ON
AND W1.05  ; OPERATION INDIVIDUAL SELECT
OUT 4603.03  ; 11ST_UNIT HOME POSITION PB
OUT 4603.04  ; 11ST_UNIT HOME POSITION PB PLUSE

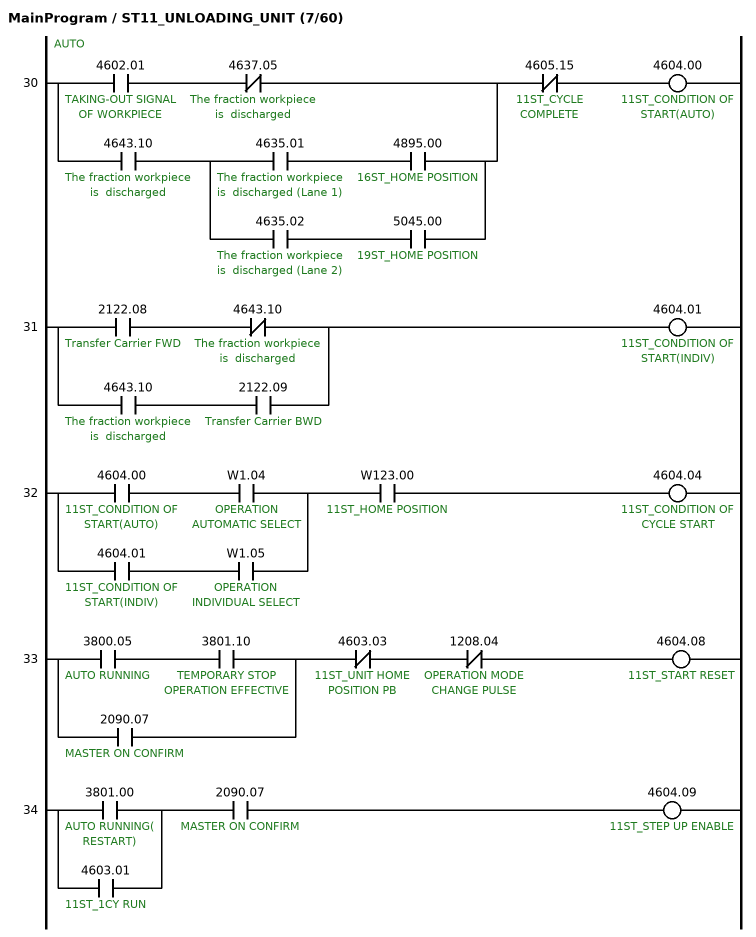
; rung 30: AUTO
LD 4602.01  ; TAKING-OUT SIGNAL OF WORKPIECE
ANDNOT 4637.05  ; The fraction workpiece is  discharged
LD 4643.10  ; The fraction workpiece is  discharged
LD 4635.01  ; The fraction workpiece is  discharged (Lane 1)
AND 4895.00  ; 16ST_HOME POSITION
LD 4635.02  ; The fraction workpiece is  discharged (Lane 2)
AND 5045.00  ; 19ST_HOME POSITION
ORLD
ANDLD
ORLD
ANDNOT 4605.15  ; 11ST_CYCLE COMPLETE
OUT 4604.00  ; 11ST_CONDITION OF START(AUTO)
; rung 31
LD 2122.08  ; Transfer Carrier FWD
ANDNOT 4643.10  ; The fraction workpiece is  discharged
LD 4643.10  ; The fraction workpiece is  discharged
AND 2122.09  ; Transfer Carrier BWD
ORLD
OUT 4604.01  ; 11ST_CONDITION OF START(INDIV)
; rung 32
LD 4604.00  ; 11ST_CONDITION OF START(AUTO)
AND W1.04  ; OPERATION AUTOMATIC SELECT
LD 4604.01  ; 11ST_CONDITION OF START(INDIV)
AND W1.05  ; OPERATION INDIVIDUAL SELECT
ORLD
AND W123.00  ; 11ST_HOME POSITION
OUT 4604.04  ; 11ST_CONDITION OF CYCLE START
; rung 33
LD 3800.05  ; AUTO RUNNING
AND 3801.10  ; TEMPORARY STOP OPERATION EFFECTIVE
OR 2090.07  ; MASTER ON CONFIRM
ANDNOT 4603.03  ; 11ST_UNIT HOME POSITION PB
ANDNOT 1208.04  ; OPERATION MODE CHANGE PULSE
OUT 4604.08  ; 11ST_START RESET
; rung 34
LD 3801.00  ; AUTO RUNNING(RESTART)
OR 4603.01  ; 11ST_1CY RUN
AND 2090.07  ; MASTER ON CONFIRM
OUT 4604.09  ; 11ST_STEP UP ENABLE

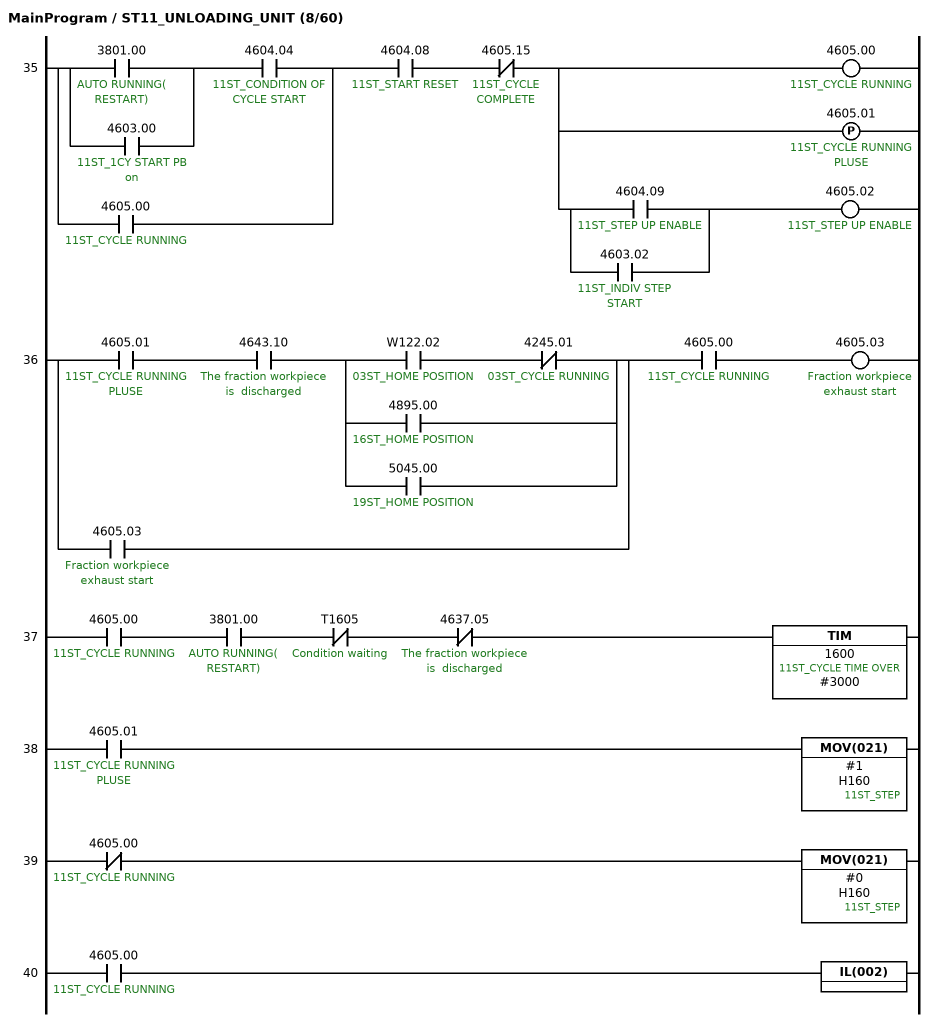
; rung 35
LD 3801.00  ; AUTO RUNNING(RESTART)
OR 4603.00  ; 11ST_1CY START PB on
AND 4604.04  ; 11ST_CONDITION OF CYCLE START
OR 4605.00  ; 11ST_CYCLE RUNNING
AND 4604.08  ; 11ST_START RESET
ANDNOT 4605.15  ; 11ST_CYCLE COMPLETE
OUT 4605.00  ; 11ST_CYCLE RUNNING
DIFU(013) 4605.01  ; 11ST_CYCLE RUNNING PLUSE
LD 4604.09  ; 11ST_STEP UP ENABLE
OR 4603.02  ; 11ST_INDIV STEP START
ANDLD
OUT 4605.02  ; 11ST_STEP UP ENABLE
; rung 36
LD 4605.01  ; 11ST_CYCLE RUNNING PLUSE
AND 4643.10  ; The fraction workpiece is  discharged
LD W122.02  ; 03ST_HOME POSITION
ANDNOT 4245.01  ; 03ST_CYCLE RUNNING
OR 4895.00  ; 16ST_HOME POSITION
OR 5045.00  ; 19ST_HOME POSITION
ANDLD
OR 4605.03  ; Fraction workpiece exhaust start
AND 4605.00  ; 11ST_CYCLE RUNNING
OUT 4605.03  ; Fraction workpiece exhaust start
; rung 37
LD 4605.00  ; 11ST_CYCLE RUNNING
AND 3801.00  ; AUTO RUNNING(RESTART)
ANDNOT T1605  ; Condition waiting
ANDNOT 4637.05  ; The fraction workpiece is  discharged
TIM 1600 #3000  ; 11ST_CYCLE TIME OVER
; rung 38
LD 4605.01  ; 11ST_CYCLE RUNNING PLUSE
MOV(021) #1 H160  ; 11ST_STEP
; rung 39
LDNOT 4605.00  ; 11ST_CYCLE RUNNING
MOV(021) #0 H160  ; 11ST_STEP
; rung 40
LD 4605.00  ; 11ST_CYCLE RUNNING
IL(002)

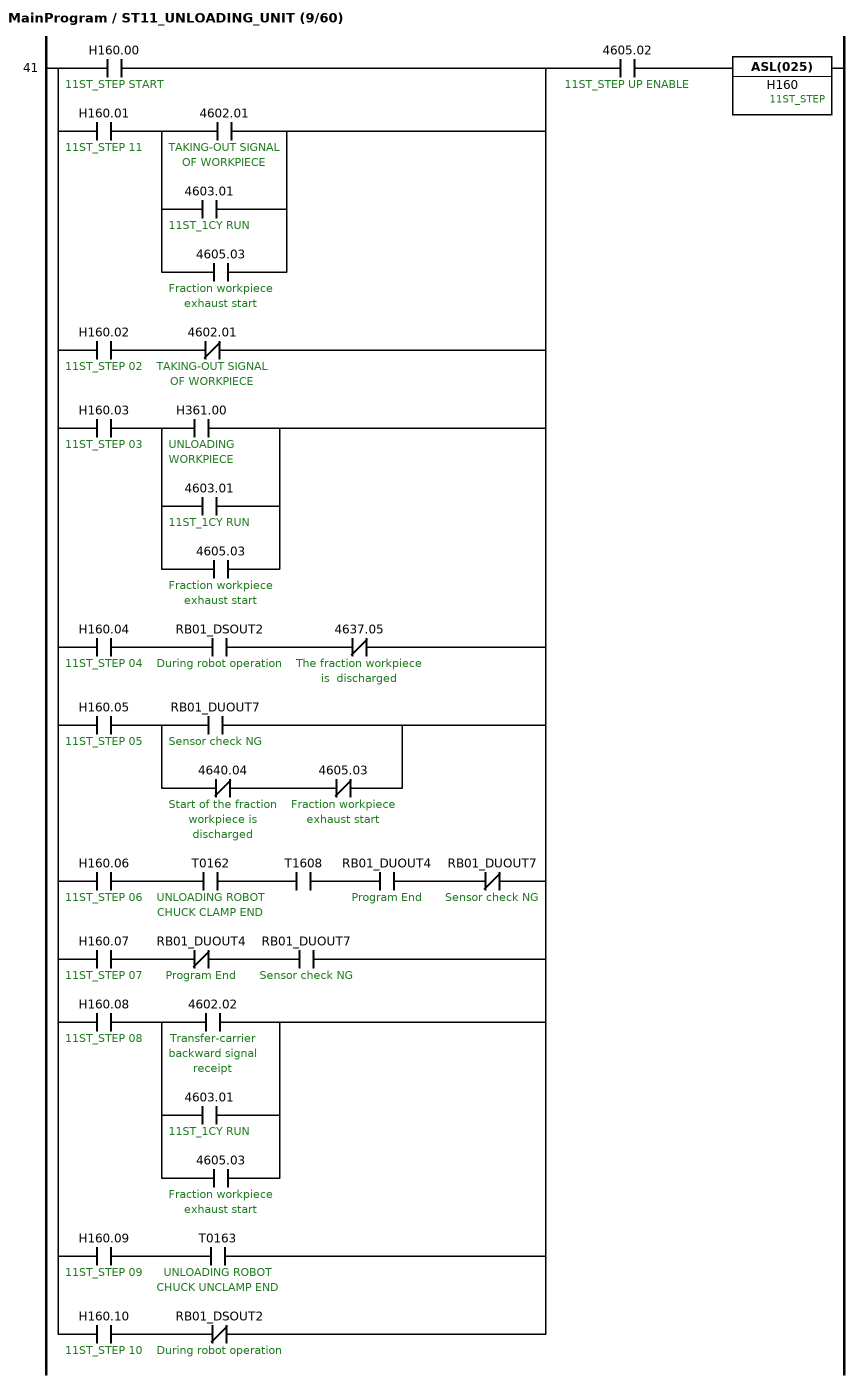
; rung 41
LD H160.00  ; 11ST_STEP START
LD H160.01  ; 11ST_STEP 11
LD 4602.01  ; TAKING-OUT SIGNAL OF WORKPIECE
OR 4603.01  ; 11ST_1CY RUN
OR 4605.03  ; Fraction workpiece exhaust start
ANDLD
ORLD
LD H160.02  ; 11ST_STEP 02
ANDNOT 4602.01  ; TAKING-OUT SIGNAL OF WORKPIECE
ORLD
LD H160.03  ; 11ST_STEP 03
LD H361.00  ; UNLOADING WORKPIECE
OR 4603.01  ; 11ST_1CY RUN
OR 4605.03  ; Fraction workpiece exhaust start
ANDLD
ORLD
LD H160.04  ; 11ST_STEP 04
AND RB01_DSOUT2  ; During robot operation
ANDNOT 4637.05  ; The fraction workpiece is  discharged
ORLD
LD H160.05  ; 11ST_STEP 05
LD RB01_DUOUT7  ; Sensor check NG
LDNOT 4640.04  ; Start of the fraction workpiece is discharged
ANDNOT 4605.03  ; Fraction workpiece exhaust start
ORLD
ANDLD
ORLD
LD H160.06  ; 11ST_STEP 06
AND T0162  ; UNLOADING ROBOT CHUCK CLAMP END
AND T1608
AND RB01_DUOUT4  ; Program End
ANDNOT RB01_DUOUT7  ; Sensor check NG
ORLD
LD H160.07  ; 11ST_STEP 07
ANDNOT RB01_DUOUT4  ; Program End
AND RB01_DUOUT7  ; Sensor check NG
ORLD
LD H160.08  ; 11ST_STEP 08
LD 4602.02  ; Transfer-carrier backward signal receipt
OR 4603.01  ; 11ST_1CY RUN
OR 4605.03  ; Fraction workpiece exhaust start
ANDLD
ORLD
LD H160.09  ; 11ST_STEP 09
AND T0163  ; UNLOADING ROBOT CHUCK UNCLAMP END
ORLD
LD H160.10  ; 11ST_STEP 10
ANDNOT RB01_DSOUT2  ; During robot operation
ORLD
AND 4605.02  ; 11ST_STEP UP ENABLE
ASL(025) H160  ; 11ST_STEP

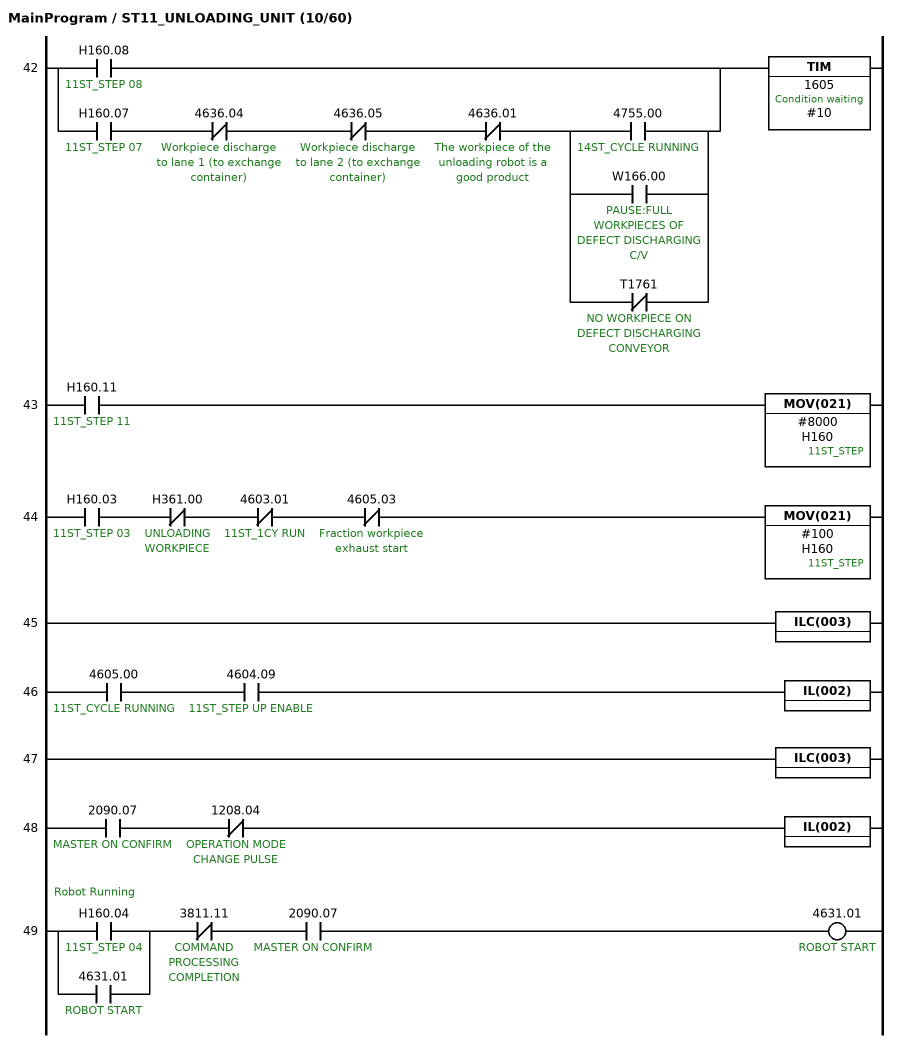
; rung 42
LD H160.08  ; 11ST_STEP 08
LD H160.07  ; 11ST_STEP 07
ANDNOT 4636.04  ; Workpiece discharge to lane 1 (to exchange container)
ANDNOT 4636.05  ; Workpiece discharge to lane 2 (to exchange container)
ANDNOT 4636.01  ; The workpiece of the unloading robot is a good product
LD 4755.00  ; 14ST_CYCLE RUNNING
OR W166.00  ; PAUSE:FULL WORKPIECES OF DEFECT DISCHARGING C/V
ORNOT T1761  ; NO WORKPIECE ON DEFECT DISCHARGING CONVEYOR
ANDLD
ORLD
TIM 1605 #10  ; Condition waiting
; rung 43
LD H160.11  ; 11ST_STEP 11
MOV(021) #8000 H160  ; 11ST_STEP
; rung 44
LD H160.03  ; 11ST_STEP 03
ANDNOT H361.00  ; UNLOADING WORKPIECE
ANDNOT 4603.01  ; 11ST_1CY RUN
ANDNOT 4605.03  ; Fraction workpiece exhaust start
MOV(021) #100 H160  ; 11ST_STEP
; rung 45
ILC(003)
; rung 46
LD 4605.00  ; 11ST_CYCLE RUNNING
AND 4604.09  ; 11ST_STEP UP ENABLE
IL(002)
; rung 47
ILC(003)
; rung 48
LD 2090.07  ; MASTER ON CONFIRM
ANDNOT 1208.04  ; OPERATION MODE CHANGE PULSE
IL(002)
; rung 49: Robot Running
LD H160.04  ; 11ST_STEP 04
OR 4631.01  ; ROBOT START
ANDNOT 3811.11  ; COMMAND PROCESSING COMPLETION
AND 2090.07  ; MASTER ON CONFIRM
OUT 4631.01  ; ROBOT START

